// TIA Portal V16 export
// export: Created 2021-09-08T12:44:32.4582115Z, ExportSetting WithDefaults, DisplayName Totally Integrated Automation Portal, DisplayVersion V16 Update 3, DisplayName TIA Portal Version Control Interface, DisplayVersion V16 Update 2, DisplayName TIA Portal Openness, DisplayVersion V16 Update 3, DisplayName TIA Portal Teamcenter Gateway, DisplayVersion V16, DisplayName STEP 7 Professional, DisplayVersion V16 Update 3, DisplayName STEP 7 Safety, DisplayVersion V16, DisplayName WinCC Advanced, DisplayVersion V16 Update 3
VAR_GLOBAL   // PLC tag table "A10_DQ"
   qDP101_Start AT %Q2.0 : Bool;   // DP101 Пуск
   qDP502_Start AT %Q2.1 : Bool;   // DP502 Пуск
   qDP501_Start AT %Q2.2 : Bool;   // DP501 Пуск
   qDP801_Start AT %Q2.3 : Bool;   // DP801 Пуск
   qDP802_Start AT %Q2.4 : Bool;   // DP802 Пуск
   qDP803_Start AT %Q2.5 : Bool;   // DP803 Пуск
   qDP1001_Start AT %Q2.6 : Bool;   // DP1001 Пуск
   "Q2.7_Reserve" AT %Q2.7 : Bool;   // Резерв
   qDVM201_Open AT %Q3.0 : Bool;   // DVM201 Відкрити
   qSOV801_Open AT %Q3.1 : Bool;   // SOV801 Відкрити
   qSOV901_Open AT %Q3.2 : Bool;   // SOV901 Відкрити
   qSOV902_Open AT %Q3.3 : Bool;   // SOV902 Відкрити
   qSOV1301_Open AT %Q3.4 : Bool;   // SOV1301 Відкрити
   qSOV1302_Open AT %Q3.5 : Bool;   // SOV1302 Відкрити
   qSOV1303_Open AT %Q3.6 : Bool;   // SOV1303 Відкрити
   "Q3.7_Reserve" AT %Q3.7 : Bool;   // Резерв
   qDVA501_Open AT %Q4.0 : Bool;   // DVA501 Відкрити
   qDVA502_Open AT %Q4.1 : Bool;   // DVA502 Відкрити
   qDVA504_Open AT %Q4.2 : Bool;   // DVA504 Відкрити
   qDVA505_Open AT %Q4.3 : Bool;   // DVA505 Відкрити
   qDVA506_Open AT %Q4.4 : Bool;   // DVA506 Відкрити
   qDVA507_Open AT %Q4.5 : Bool;   // DVA507 Відкрити
   qDVA508_Open AT %Q4.6 : Bool;   // DVA508 Відкрити
   qDVA509_Open AT %Q4.7 : Bool;   // DVA509 Відкрити
   qDVA511_Open AT %Q5.0 : Bool;   // DVA511 Відкрити
   qDVA512_Open AT %Q5.1 : Bool;   // DVA512 Відкрити
   qDVA513_Open AT %Q5.2 : Bool;   // DVA513 Відкрити
   qDVA514_Open AT %Q5.3 : Bool;   // DVA514 Відкрити
   qDVA515_Open AT %Q5.4 : Bool;   // DVA515 Відкрити
   qDVA516_Open AT %Q5.5 : Bool;   // DVA516 Відкрити
   qDVA1801_Open AT %Q5.6 : Bool;   // DVA1801 Відкрити
   qMDF4 AT %Q5.7 : Bool;   // Фільтр дисковий
END_VAR
VAR_GLOBAL CONSTANT   // user constants
   "qDP-101_Start" : Int := 0;
   "qDP-502_Start" : Int := 1;
   "qDP-501_Start" : Int := 2;
   "qDP-801_Start" : Int := 3;
   "qDP-802_Start" : Int := 4;
   "qDP-803_Start" : Int := 5;
   "qDP-1001_Start" : Int := 6;
   "Q2.7_res" : Int := 7;
   "qDVM-201_Open" : Int := 8;
   "qSOV-801_Open" : Int := 9;
   "qSOV-901_Open" : Int := 10;
   "qSOV-902_Open" : Int := 11;
   "qSOV-1301_Open" : Int := 12;
   "qSOV-1302_Open" : Int := 13;
   "qSOV-1303_Open" : Int := 14;
   "Q3.7_res" : Int := 15;
   "qDVA-501_Open" : Int := 16;
   "qDVA-502_Open" : Int := 17;
   "qDVA-504_Open" : Int := 18;
   "qDVA-505_Open" : Int := 19;
   "qDVA-506_Open" : Int := 20;
   "qDVA-507_Open" : Int := 21;
   "qDVA-508_Open" : Int := 22;
   "qDVA-509_Open" : Int := 23;
   "qDVA-511_Open" : Int := 24;
   "qDVA-512_Open" : Int := 25;
   "qDVA-513_Open" : Int := 26;
   "qDVA-514_Open" : Int := 27;
   "qDVA-515_Open" : Int := 28;
   "qDVA-516_Open" : Int := 29;
   "qDVA-1801_Open" : Int := 30;
   "Q5.7_res" : Int := 31;
END_VAR
